(* if rst then *)
IF rst THEN
	piwl(rst := TRUE);
	piwl.RST := FALSE;
ELSE
	(* run PIWL controller first *)
	(* we need to check if TN = 0 and do alternative calls *)
	IF TN = 0.0 THEN
		piwl(in := IN * KP, KP := 1.0, KI := 0.0, LIM_L := LIM_L, LIM_H := LIM_H);
	ELSE
		piwl(in := IN * KP, KP := 1.0, KI := 1.0 / TN, LIM_L := LIM_L, LIM_H := LIM_H);
	END_IF;

	(* run differentiator and add_to_output *)
	diff(IN := IN, K := KP * TV);
	Y := piwl.Y + diff.out;
	(* add: output signal parts separately *)
	Y_p := piwl.Y_p;
	Y_i := piwl.Y_i;
	Y_d := diff.out;

	(* limit the output *)
	IF Y > LIM_H THEN
		Y := LIM_H;
		IF (Y_i > 0) THEN
			Y_i := LIM_H - Y_p - Y_d;
		END_IF
		LIM := TRUE;
	ELSIF Y < LIM_L THEN
		Y := LIM_L;
		IF (Y_i > 0) THEN
			Y_i := LIM_L - Y_p - Y_d;
		END_IF
		LIM := TRUE;
	ELSE
		LIM := FALSE;
	END_IF;
	
END_IF;



(* revision history
hm 13. jun. 2008 	rev 1.0
	original version

hm	25. jan 2008	rev 1.1
	multiply differential part with KP

hm	11. mar. 2009	rev 1.2
	real constants updated to new systax using dot

hm	13. nov. 2009	rev 1.3
	fixed code for negative KP

*)

END_FUNCTION_BLOCK

// A1_01A/Application/FUBs/Controller
// https://ftp.owen.ru/CoDeSys3/98_Books/oscat_basic333_ru.pdf		page 543, page 551
FUNCTION_BLOCK Controller
VAR_INPUT
	in: ctrl_input_typ;
	param: ctrl_param_typ;	
	cmd: ctrl_cmd_typ;
	cfg: UINT;
	t_move: UINT := 100;			// время на полную перестановку, сек (в текущей реализации как-то не у дел)
	t_error: UINT := 120;			// время на схождение положения крана и регулятора при регулировании
END_VAR
VAR_OUTPUT
	out: ctrl_output_typ;
	flags: ctrl_flags_typ;
END_VAR
VAR
	fub_pid: CTRL_PID;
	ton_diff: Standard.TON;
	ton_imit: Standard.TON;
END_VAR

(* Регулятор. 2 режима работы: стандартный, выход на ао
 * mode_manual - режим ручного ввода положения. управление аналоговое *)
		
IF cmd.manual_on THEN
	cmd.manual_on := FALSE;
	flags.mode_manual := TRUE;
END_IF
IF cmd.manual_off THEN
	cmd.manual_off := FALSE;
	flags.mode_manual := FALSE;
END_IF

IF cmd.imit_on THEN
	cmd.imit_on := FALSE;
	flags.mode_imit := TRUE;
	// при вкл имитации переведем пид в ручной режим на текущем уровне открытия и уставки
	in.man_value := in.im_pos_value := in.pos_value;
	in.set_value := in.act_value;
END_IF
IF cmd.imit_off THEN
	cmd.imit_off := FALSE;
	flags.mode_imit := FALSE;
END_IF

IF cmd.reset THEN
	cmd.reset := FALSE;
	flags.fail_open := FALSE;
	flags.fail_close := FALSE;
	flags.failed := FALSE;
END_IF
IF cmd.line_close THEN
	cmd.line_close := FALSE;
	IF flags.mode_imit THEN
		ton_imit.IN := TRUE;
		ton_imit.PT := REAL_TO_TIME( (UINT_TO_REAL(t_move) * in.im_pos_value/2/100)*1000 + 1);
	ELSE
		ton_imit.IN := FALSE;
		;// уставки приходится задавать снаружи (или встраивать alg_sp в пид)
	END_IF
END_IF
IF flags.mode_imit THEN
	in.pos_value := in.im_pos_value;
	// выход out_value не трогаем
	
	//IF b THEN
	ton_imit();
	//END_IF
	
	IF ton_imit.IN THEN
		in.im_pos_value := TIME_TO_REAL((ton_imit.PT - ton_imit.ET) / 1000 * 2);
	END_IF
	IF ton_imit.Q THEN
		ton_imit.IN := FALSE;
		in.im_pos_value := 0;
	END_IF
END_IF

fub_pid.ACT := in.act_value;
fub_pid.SET := in.set_value;
fub_pid.SUP := param.dead_zone;
fub_pid.OFS := param.offset;
fub_pid.M_I := in.man_value;
fub_pid.LL := param.min_out;
fub_pid.LH := param.max_out;
fub_pid.KP := param.k_p;
fub_pid.TN := param.t_i;
fub_pid.TV := param.t_d;
fub_pid.MAN := flags.mode_manual OR flags.mode_imit;
fub_pid();
out.err_value := fub_pid.DIFF;
out.out_value := fub_pid.Y;
out.p_part := fub_pid.Y_p;
out.i_part := fub_pid.Y_i;
out.d_part := fub_pid.Y_d;

flags.mode_dist := in.di_dist;
in.hyst_value := LIMIT(0.0, in.hyst_value, 5.0);
IF cfg.discrete_input THEN
	flags.open := in.di_open;
	flags.closed := in.di_closed;
ELSE
	flags.closed := in.pos_value <= in.hyst_value;
	flags.open := in.pos_value >= (100.0 - in.hyst_value);
END_IF

// Формирование команд дискретного управления регулирующим клапаном
flags.block_ao := NOT flags.mode_dist OR flags.mode_discrete OR flags.mode_manual OR flags.mode_imit;//cmd.line_close;
flags.ready := NOT in.di_fail AND flags.mode_dist AND NOT flags.block_ao; //исправим на NOT block_ao, потому что вообще нелогично

// Формирование сигнала «Неисправность регулирующего клапана»
ton_diff(IN := (param.discrepancy > 0.0 AND t_error > 0) AND_THEN ABS(in.pos_value - out.out_value) > (param.discrepancy + in.hyst_value) AND NOT flags.block_ao, PT := UDINT_TO_TIME(UINT_TO_UDINT(t_error) * 1000));
IF NOT flags.failed AND_THEN (in.di_fail OR ton_diff.Q OR flags.fail_open OR flags.fail_close) THEN
	flags.failed := TRUE;
	flags.mode_manual := TRUE;
END_IF

END_FUNCTION_BLOCK

// A1_01A/Application/Oscat/DEAD_ZONE
FUNCTION DEAD_ZONE : REAL
VAR_INPUT
	X : REAL;
	L : REAL;
END_VAR


(*
version 1.2	11. mar. 2009
programmer 	hugo
tested by		oscat

dead_zone2 is a linear transfer function which follows a linear function except for x is close to 0.
Y = X if abs(x) > L otherwise its 0.

*)

IF ABS(x) > L THEN
	dead_zone := X;
ELSE
	DEAD_ZONE := 0.0;
END_IF;

(* revision history
hm	12. feb. 2007	rev 1.0
	original version

hm	14. jun. 2008	rev 1.1
	improved performance

hm	11. mar. 2009	rev 1.2
	real constants updated to new systax using dot

*)

END_FUNCTION

// A1_01A/Application/Oscat/CTRL_PID
FUNCTION_BLOCK CTRL_PID
VAR_INPUT
	ACT : REAL;			// Значение регулируемой величины
	SET : REAL;			// Значение уставки
	SUP : REAL;			// Зона нечувствительности
	OFS : REAL;			// Смещение
	M_I : REAL;			// Значение ручного ввода
	MAN : BOOL;			// Сигнал ручного ввода
	RST : BOOL;			// Сигнал обнуления И-составляющей
	KP : REAL := 1.0;
	TN : REAL := 1.0;
	TV : REAL := 1.0;
	LL : REAL := -1000.0;	// Нижний предел управляющего сигнала
	LH : REAL := 1000.0;	// Верхний предел управляющего сигнала
END_VAR
VAR_OUTPUT
	Y : REAL;			// Величина управляющего воздействия
	Y_p : REAL;
	Y_i : REAL;
	Y_d : REAL;
	DIFF : REAL;		// Сигнал рассогласования
	LIM : BOOL;			// Флаг «достигнут предел для Y»
END_VAR
VAR
	pid : FT_PIDWL;
	co : CTRL_OUT;
END_VAR



(*
version 2.0	30. jun. 2008
programmer 	hugo
tested by	oscat

FT_PI is a PI controller with manual functionality.
The PID controller works according to the fomula Y = e *(KP+ KI * INTEG(e) ) + offset, while e = set_point - actual.
a rst will reset all internal data, while a switch to manual will cause the controller to follow the function Y = manual_in + offset.
limit_h and Limit_l set the possible output range of Y.
the output flags lim will signal that the output limits are active.

*)

DIFF := CTRL_IN(SET, ACT, SUP);
pid(in := DIFF, kp := KP, tn := TN, tv := TV, lim_l := LL, lim_h := LH, rst := RST);
co(ci := pid.Y, OFFSET := OFS, man_in := M_I, lim_l := LL, lim_h := LH, MANUAL := MAN);
Y := co.Y;
LIM := co.LIM;

Y_p := pid.Y_p;
Y_i := pid.Y_i;
Y_d := pid.Y_d;

(* revision history

hm 1.12.2006	 	rev 1.1
	changed algorithm to trapezregel for higher accuracy.

hm 3.1.2007		rev 1.2
	added integ_band to select when the integrator is active.

hm	3.3.2007		rev 1.3
	added default values to inputs KP, TN, TV, LIMIT_L und LIMIT_H.

hm 31.oct 2007	rev 1.4
	total rewrite of the module to avoid failures when one of the limits is 0

hm	3.11.2007	rev 1.5
	added noise input to filter noise
	added output diff
	set limit output false when output is within limits
	overfolw was not set correctly

hm	5. jan 2008	rev 1.6
	improved code for better performance
*)

END_FUNCTION_BLOCK

// A1_01A/Application/Oscat/CTRL_IN
FUNCTION CTRL_IN : REAL
VAR_INPUT
	SET_POINT, ACTUAL, NOISE : REAL;
END_VAR


(*
version 1.0	2. jun 2008
programmer 	hugo
tested by		tobias


*)

(* calculate the process error DIFF *)
CTRL_IN := DEAD_ZONE(SET_POINT - ACTUAL, NOISE);


(* revision history
hm 	2. jun. 2008 	rev 1.0
	original version

*)

END_FUNCTION

// A1_01A/Application/Oscat/FT_PIWL
FUNCTION_BLOCK FT_PIWL
VAR_INPUT
	IN : REAL;
	KP : REAL := 1.0;
	KI : REAL := 1.0;
	LIM_L : REAL := -1.0E38;
	LIM_H : REAL := 1.0E38;
	RST : BOOL;
END_VAR
VAR_OUTPUT
	Y : REAL;
	Y_p : REAL;
	Y_i : REAL;
	LIM : BOOL;
END_VAR
VAR
	init: BOOL;
	tx: DWORD;
	tc : REAL;
	t_last: DWORD;
	in_last : REAL;
	i: REAL;
	p: REAL;
END_VAR

(*
version 1.3	11. mar. 2009
programmer 	hugo
tested by		oscat

FT_PIWL is a PI controller.
The PID controller works according to the fomula Y = IN *(KP+ KI * INTEG(e) ).
a rst will reset the integrator to 0
lim_h and Lim_l set the possible output range of the controller.
the output flag lim will signal that the output limits are active.
the integrator ist equipped with anti wind-up circuitry which limits trhe total output ranke to lim_l and lim_h

default values for KP = 1, KI = 1, ILIM_L = -1E37, iLIM_H = +1E38.
*)

(* initialize at power_up *)
IF NOT init OR RST THEN
	init := TRUE;
	in_last := in;
	t_last := T_PLC_US();
	i := 0.0;
	tc := 0.0;
ELSE
	(* read last cycle time in Microseconds *)
	tx := T_PLC_US();
	tc := DWORD_TO_REAL(tx - t_last);
	t_last := tx;

	(* calculate proportional part *)
	p := KP * IN;

	(* run integrator *)
	i := (IN + in_last) * 5.0E-7 * KI * tc + i;
	in_last := IN;

	(* calculate output Y *)
	Y := p + i;

	(* check output for limits *)
	IF Y >= LIM_H THEN
		Y := LIM_H;
		IF ki <> 0.0 THEN
			i := LIM_H - p;
		ELSE
			i := 0.0;
		END_IF;
		LIM := TRUE;
	ELSIF Y <= LIM_L THEN
		Y := LIM_L;
		IF ki <> 0.0 THEN
			i := LIM_L - p;
		ELSE
			i := 0.0;
		END_IF;
		LIM := TRUE;
	ELSE
		LIM := FALSE;
	END_IF;
	
	(* add: output signal parts separately *)
	Y_p := p;
	Y_i := i;
END_IF;




(* revision history
hm 13. jun. 2008 	rev 1.0
	original version

hm	27. oct. 2008	rev 1.1
	integrator will not be adjusted when ki = 0

hm	25. jan 2009	rev 1.2
	module will also work with negative K

hm	11. mar. 2009	rev 1.3
	real constants updated to new systax using dot

*)

END_FUNCTION_BLOCK

// A1_01A/Application/Oscat/FT_DERIV
FUNCTION_BLOCK FT_DERIV
VAR_INPUT
	in : REAL;
	K : REAL := 1.0;
	run : BOOL := TRUE;
END_VAR
VAR_OUTPUT
	out : REAL;
END_VAR
VAR
	old: REAL;
	tx: DWORD;
	last: DWORD;
	init: BOOL;
	tc: REAL;
END_VAR


(*
version 1.5	11. mar. 2009
programmer 	hugo
tested by		oscat

FT_deriv calculates the derivate over the signal "in" with Faktor "K".
a run input enables or stops the calculation, if left unconnected its true and therfore the calculation is executed.
if K is not specified the default is 1.

*)

(* read system time *)
tx := T_PLC_US();
tc := DWORD_TO_REAL(tx - last);
last := tx;

(* init on first startup *)
IF NOT init THEN
	init := TRUE;
	old := in;
ELSIF run AND tc > 0.0 THEN
	out := (in - old) / tc * 1000000.0 * K;
	old := in;
ELSE
	out := 0.0;
END_IF;



(*
hm 3.1.2007			rev 1.1
	added init code for startup
	set the default for K to 1

hm	15. sep 2007	rev 1.2
	replaced Time() with T_PLC_US for compatibility and performance reasons
	increased accuracy and work in microseconds internally

hm 29 oct 2007	rev 1.3
	prohibit calculation when tx - last = 0 to avoid division by 0 and increase accuracy on fast systems

hm	6. nov. 2008	rev 1.4
	improved performance

hm	11. mar. 2009	rev 1.5
	inproved code
*)

END_FUNCTION_BLOCK

// A1_01A/Application/FUBs/LineMeteringRLT
FUNCTION_BLOCK LineMeteringRLT	// Алгоритм нитки расхода
VAR_INPUT
	num_v_in, num_v_out: UINT;	// номера кранов из массива на входе/выходе этой нитки
	param: line_param_f_typ;
	cmd: line_cmd_typ;			// прямые команды управления 
	a_in: line_act_in;			// внешнее алгоритмическое управление
	a_out: line_act_out;		// результат исполнения
	flow_online: BOOL;			// расходомер на связи, расход актуален
	busy: BOOL;					// нитка занята в алгоритме
	a_to: USINT;				// номер нитки, в которую была выдана команда
END_VAR
VAR_OUTPUT
	flags: line_flags_f_typ;
END_VAR
VAR
END_VAR

IF cmd.block_on THEN
	cmd.block_on := FALSE;
	flags.mode_block := TRUE;
END_IF
IF cmd.block_off THEN
	cmd.block_off := FALSE;
	flags.mode_block := FALSE;
END_IF
IF cmd.manual_on THEN
	cmd.manual_on := FALSE;
	flags.mode_manual := TRUE;
END_IF
IF cmd.manual_off THEN
	cmd.manual_off := FALSE;
	flags.mode_manual := FALSE;
END_IF
IF cmd.reset THEN
	cmd.reset := FALSE;
	flags.failed := FALSE;
	flags.fail_block := FALSE;
END_IF
IF (flags.mode_block AND (a_in.a_cmd > 0 OR cmd.open OR cmd.close)) THEN
	a_in.a_cmd := en_line_action.LA_NONE;
	a_in.a_from := -1;
	cmd.open := FALSE;
	cmd.close := FALSE;
	flags.fail_block := TRUE;
END_IF

IF num_v_in < COUNT_VALVE AND num_v_out < COUNT_VALVE THEN
	flags.err_num := FALSE;
	flags.open := sys_valve[num_v_in].v_state = RLTAB.en_valve_state.VALVESTT_OPEN AND sys_valve[num_v_out].v_state = RLTAB.en_valve_state.VALVESTT_OPEN;
	flags.closed := sys_valve[num_v_in].v_state = RLTAB.en_valve_state.VALVESTT_CLOSED AND sys_valve[num_v_out].v_state = RLTAB.en_valve_state.VALVESTT_CLOSED;
	flags.ready := (sys_valve[num_v_in].flags.ready AND sys_valve[num_v_out].flags.ready) AND NOT flags.mode_block;
	// T6.1,141 Формирование сигнала о неисправности линии редуцирования
	// VALVE: flags.ready := (v_mode > MODE_BUTTON) AND NOT flags.mode_block AND NOT (flags.cv_fail OR flags.fail_open OR flags.fail_close);
	IF flags.open AND NOT flags.ready AND NOT flags.mode_reserve THEN
		flags.failed := TRUE;
	END_IF
	
	IF flags.mode_manual THEN
		param.flow_actual := param.flow_manual;
	END_IF
	IF flags.open AND param.flow_lo <> param.flow_hi THEN
		IF param.flow_actual < (param.flow_lo - param.flow_hyst) THEN
			flags.flow_lo := TRUE;
			flags.flow_ok := FALSE;
		ELSIF param.flow_actual > (param.flow_lo + param.flow_hyst) THEN
			flags.flow_lo := FALSE;
			flags.flow_ok := TRUE;
		END_IF
		IF param.flow_actual > (param.flow_hi + param.flow_hyst) THEN
			flags.flow_hi := TRUE;
			flags.flow_ok := FALSE;
		ELSIF param.flow_actual < (param.flow_hi - param.flow_hyst) THEN
			flags.flow_hi := FALSE;
			flags.flow_ok := TRUE;
		END_IF
	ELSE
		flags.flow_lo := FALSE;
		flags.flow_ok := FALSE;
		flags.flow_hi := FALSE;
	END_IF
		
	// лучше использовать эти команды a_in для внешнего алгоритмического управления, т.к. в них встроена защита от busy
	IF a_in.a_cmd > 0 THEN
		a_out.done := FALSE;
		IF a_out.result <> en_line_action.LA_BUSY (*AND NOT flags.mode_block*) THEN
			a_out.a_orig := a_in.a_cmd;
			//a_in.a_cmd := en_line_action.LA_NONE;
			a_out.a_from := a_in.a_from;
			//a_in.a_from := -1;
			CASE a_out.a_orig OF
				en_line_action.LA_OPEN:
					cmd.open := TRUE;
				en_line_action.LA_CLOSE:
					cmd.close := TRUE;
			END_CASE
			a_out.result := en_line_action.LA_BUSY;
		END_IF
		a_in.a_cmd := en_line_action.LA_NONE;
		a_in.a_from := -1;
	END_IF
	IF a_out.result = en_line_action.LA_BUSY THEN
		CASE a_out.a_orig OF
			en_line_action.LA_OPEN:
				IF flags.ready THEN
					IF flags.open THEN
						a_out.result := en_line_action.LA_OPEN;
						a_out.done := TRUE;
					END_IF
				ELSE
					a_out.result := en_line_action.LA_ERROR;
					a_out.done := TRUE;
				END_IF
				
			en_line_action.LA_CLOSE:
				IF flags.ready THEN
					IF flags.closed THEN
						a_out.result := en_line_action.LA_CLOSE;
						a_out.done := TRUE;
					END_IF
				ELSE
					a_out.result := en_line_action.LA_ERROR;
					a_out.done := TRUE;
				END_IF
				
		END_CASE
	END_IF
	
	IF cmd.open THEN
		cmd.open := FALSE;
		sys_valve[num_v_in].cmd.open := TRUE;
		sys_valve[num_v_out].cmd.open := TRUE;
	END_IF
	IF cmd.close THEN
		cmd.close := FALSE;
		sys_valve[num_v_in].cmd.close := TRUE;
		sys_valve[num_v_out].cmd.close := TRUE;
	END_IF
ELSE
	flags.err_num := TRUE;
	flags.open := FALSE;
	flags.closed := FALSE;
	flags.ready := FALSE;
	a_in.a_cmd := en_line_action.LA_NONE;
	a_in.a_from := -1;
	cmd.open := FALSE;
	cmd.close := FALSE;
END_IF

METHOD Init
VAR_INPUT
	value: BOOL;
END_VAR
THIS^.flags.mode_reserve := value;
END_METHOD

METHOD _set_mr
VAR_INPUT
	value: BOOL;
END_VAR
THIS^.flags.mode_reserve := value;
END_METHOD

END_FUNCTION_BLOCK

// A1_01A/Application/FUBs/LineReducingRLT
FUNCTION_BLOCK LineReducingRLT	// Алгоритм нитки редуцирования
VAR_INPUT
	num_ctrl: UINT;				// номер ПИДа на этой нитки
	num_v_in, num_v_out: UINT;	// номера кранов из массива на входе/выходе этой нитки
	cmd: line_cmd_typ;			// прямые команды управления 
	a_in: line_act_in;			// внешнее алгоритмическое управление
	a_out: line_act_out;		// результат исполнения
	busy: BOOL;					// нитка занята в алгоритме
	a_to: USINT;				// номер нитки, в которую была выдана команда
END_VAR
VAR_OUTPUT
	flags: line_flags_r_typ;
END_VAR
VAR
END_VAR

IF cmd.block_on THEN
	cmd.block_on := FALSE;
	flags.mode_block := TRUE;
END_IF
IF cmd.block_off THEN
	cmd.block_off := FALSE;
	flags.mode_block := FALSE;
END_IF
IF cmd.reset THEN
	cmd.reset := FALSE;
	flags.failed := FALSE;
	flags.fail_block := FALSE;
END_IF
IF (flags.mode_block AND (a_in.a_cmd > 0 OR cmd.open OR cmd.close)) THEN
	a_in.a_cmd := en_line_action.LA_NONE;
	a_in.a_from := -1;
	cmd.open := FALSE;
	cmd.close := FALSE;
	flags.fail_block := TRUE;
END_IF

IF num_v_in < COUNT_VALVE AND num_ctrl < CFGCONST.COUNT_LINES AND num_v_out < COUNT_VALVE THEN
	flags.err_num := FALSE;
	flags.open := sys_valve[num_v_in].v_state = RLTAB.en_valve_state.VALVESTT_OPEN AND sys_valve[num_v_out].v_state = RLTAB.en_valve_state.VALVESTT_OPEN;
	flags.closed := sys_valve[num_v_in].v_state = RLTAB.en_valve_state.VALVESTT_CLOSED AND pid[num_ctrl].flags.closed AND sys_valve[num_v_out].v_state = RLTAB.en_valve_state.VALVESTT_CLOSED;
	flags.ready := (sys_valve[num_v_in].flags.ready AND pid[num_ctrl].flags.ready AND sys_valve[num_v_out].flags.ready) AND NOT flags.mode_block;
	// T6.1,141 Формирование сигнала о неисправности линии редуцирования
	// VALVE: flags.ready := (v_mode > MODE_BUTTON) AND NOT flags.mode_block AND NOT (flags.cv_fail OR flags.fail_open OR flags.fail_close);
	IF flags.open AND NOT flags.ready AND NOT flags.mode_reserve THEN
		flags.failed := TRUE;
	END_IF
	
	// лучше использовать эти команды a_in для внешнего алгоритмического управления, т.к. в них встроена защита от busy
	IF a_in.a_cmd > 0 THEN
		a_out.done := FALSE;
		IF a_out.result <> en_line_action.LA_BUSY (*AND NOT flags.mode_block*) THEN
			a_out.a_orig := a_in.a_cmd;
			//a_in.a_cmd := en_line_action.LA_NONE;
			a_out.a_from := a_in.a_from;
			//a_in.a_from := -1;
			CASE a_out.a_orig OF
				en_line_action.LA_OPEN:
					cmd.open := TRUE;
				en_line_action.LA_CLOSE:
					cmd.close := TRUE;
			END_CASE
			a_out.result := en_line_action.LA_BUSY;
		END_IF
		a_in.a_cmd := en_line_action.LA_NONE;
		a_in.a_from := -1;
	END_IF
	IF a_out.result = en_line_action.LA_BUSY THEN
		CASE a_out.a_orig OF
			en_line_action.LA_OPEN:
				IF flags.ready THEN
					IF flags.open THEN
						a_out.result := en_line_action.LA_OPEN;
						a_out.done := TRUE;
					END_IF
				ELSE
					a_out.result := en_line_action.LA_ERROR;
					a_out.done := TRUE;
				END_IF
				
			en_line_action.LA_CLOSE:
				IF flags.ready THEN
					IF flags.closed THEN
						a_out.result := en_line_action.LA_CLOSE;
						a_out.done := TRUE;
					END_IF
				ELSE
					a_out.result := en_line_action.LA_ERROR;
					a_out.done := TRUE;
				END_IF
				
		END_CASE
	END_IF
	
	IF cmd.open THEN
		cmd.open := FALSE;
		sys_valve[num_v_in].cmd.open := TRUE;
		pid[num_ctrl].cmd.manual_off := TRUE;
		sys_valve[num_v_out].cmd.open := TRUE;
	END_IF
	IF cmd.close THEN
		cmd.close := FALSE;
		sys_valve[num_v_in].cmd.close := TRUE;
		pid[num_ctrl].cmd.line_close := TRUE;
		pid[num_ctrl].cmd.manual_on := TRUE;
		sys_valve[num_v_out].cmd.close := TRUE;
	END_IF
ELSE
	flags.err_num := TRUE;
	flags.open := FALSE;
	flags.closed := FALSE;
	flags.ready := FALSE;
	a_in.a_cmd := en_line_action.LA_NONE;
	a_in.a_from := -1;
	cmd.open := FALSE;
	cmd.close := FALSE;
END_IF

METHOD Init
VAR_INPUT
	value: BOOL;
END_VAR
THIS^.flags.mode_reserve := value;
END_METHOD

METHOD _set_mr
VAR_INPUT
	value: BOOL;
END_VAR
THIS^.flags.mode_reserve := value;
END_METHOD

END_FUNCTION_BLOCK

// A1_01A/Application/FUBs/LineGroupRLT
FUNCTION_BLOCK LineGroupRLT			// Алгоритм управления группой ниток по аналогам БАКСа
VAR_INPUT							// поддерживает LineReducingRLT и LineMeteringRLT без доработок через объявление в GVL
	lines: ARRAY [0..COUNT_LINES-1] OF UINT;	// номера ниток в группе 0..max-1
	count: UINT := CFGCONST.COUNT_LINES;		// кол-во ниток, макс все в одной группе 
	cmd: line_cmd_grp_typ;
	
	new_res_line: UINT;				// новая резервная нитка
	lines_needed: USINT;			// сколько ниток требуется
	t_change: UINT := 30;			// время на перестановку линии, сек
	enable: BOOL;
	automatic: BOOL;				// включен автоматический режим
	stop_now: BOOL;					// немедленно все закрыть
END_VAR
VAR_OUTPUT
	lines_at_work: USINT;			// столько ниток в работе
	old_res_line: UINT;				// текущая резервная нитка
	// алгоритм: смена резервной нитки
	line_reserve_want: BOOL;		// алгоритм хочет запустится, но нитки еще заняты другим
	line_reserve_run: BOOL;			// алгоритм работает
	line_reserve_fail: BOOL;		// авария алгоритма
	// алгоритм: переключение ниток по аварии
	line_fault_block: BOOL;			// алгоритм заблокирован
	line_fault_want: BOOL;
	line_fault_run: BOOL;
	line_fault_fail: BOOL;
	// алгоритм: управление нитками по расходу
	line_flow_block: BOOL;
	line_flow_want: BOOL;
	line_flow_run: BOOL;
	line_flow_no_open: BOOL;		// нет нитки для открытия
	line_flow_no_close: BOOL;		// нет нитки для закрытия
END_VAR
VAR
	ton_res: Standard.TON;
	ton_fault: Standard.TON;
	ton_flow: Standard.TON;
	i, j, n: USINT;
	b, v: BOOL;
END_VAR

IF NOT enable THEN
	RETURN;
END_IF
IF count > CFGCONST.COUNT_LINES THEN
	count := CFGCONST.COUNT_LINES;
END_IF
//	в принципе эти алгоритмы подходят для любых ниток с похожим интерейсом. можно переделать через него...
//	управление: count, new_res_line, lines_needed, у ниток: cmd, flags

IF cmd.block_fault_on THEN
	cmd.block_fault_on := FALSE;
	line_fault_block := TRUE;
END_IF
IF cmd.block_fault_off THEN
	cmd.block_fault_off := FALSE;
	line_fault_block := FALSE;
END_IF
IF cmd.block_flow_on THEN
	cmd.block_flow_on := FALSE;
	line_flow_block := TRUE;
END_IF
IF cmd.block_flow_off THEN
	cmd.block_flow_off := FALSE;
	line_flow_block := FALSE;
END_IF
IF stop_now THEN
	line_fault_block := TRUE;
	line_flow_block := TRUE;
END_IF

IF cmd.close THEN
	IF NOT line_reserve_run AND NOT line_reserve_run AND NOT line_flow_run THEN
		cmd.close := FALSE;
		FOR i := 0 TO CFGCONST.COUNT_LINES-1 DO
			line[i].a_in.a_cmd := en_line_action.LA_CLOSE;
			line[i].a_in.a_from := 0;
		END_FOR
	END_IF
END_IF
IF cmd.reset THEN
	cmd.reset := FALSE;
	line_reserve_fail := FALSE;
	line_fault_fail := FALSE;
	line_flow_no_open := FALSE;
	line_flow_no_close := FALSE;
	FOR i := 0 TO CFGCONST.COUNT_LINES-1 DO
		line[i].cmd.reset := TRUE;
	END_FOR
END_IF

// ПОКА ЧТО оставим захардкоженные линии 6 штук. подумать как присвоить их потом
lines_at_work := 0;
FOR i := 0 TO CFGCONST.COUNT_LINES-1 DO
	line[i]();
	lines_at_work := lines_at_work + BOOL_TO_USINT(line[i].flags.open);
END_FOR

// общее: начинаем общий алгоритм если ничего другого не исполняется и если нет блока
// но если уже работает, должен дойти до конца

// Алгоритм: смена резервной нитки
IF new_res_line <> old_res_line AND NOT line_reserve_fail AND NOT line_reserve_run THEN	// "AND NOT line_reserve_run" здесь не особо обязателен, т.к. есть в IF ниже. но "заход" тогда все равно пустой получается
	IF automatic AND NOT stop_now AND NOT line_fault_run AND NOT line_flow_run THEN
		//IF NOT line_reserve_run THEN
			line_reserve_run := TRUE;
			line_reserve_want := FALSE;
		//END_IF
	ELSE
		line_reserve_want := TRUE;
	END_IF
ELSE
	line_reserve_want := FALSE;
END_IF
ton_res(IN := line_reserve_run, PT := UDINT_TO_TIME(UINT_TO_UDINT(t_change) * 1000));
IF line_reserve_run THEN
	IF NOT line[old_res_line].flags.ready OR NOT line[new_res_line].flags.ready OR ton_res.Q THEN		// flags.failed ? в ready включены аварии кранов, но оно сбрасывается само
		// в данном случае ошибки кранов включены в флаг ready, поэтому так норм
		line_reserve_run := FALSE;
		//old_res_line := new_res_line;
		line_reserve_fail := TRUE;
	ELSIF line[old_res_line].flags.closed AND line[new_res_line].flags.closed THEN
		line_reserve_run := FALSE;
		line[old_res_line]._set_mr(FALSE);
		line[new_res_line]._set_mr(TRUE);
		old_res_line := new_res_line;
	ELSE
		// откроем новую линию, затем закроем старую. после завершения поменяем статусы
		IF NOT line[old_res_line].flags.open THEN
			line[old_res_line].a_in.a_cmd := en_line_action.LA_OPEN;
			line[old_res_line].a_in.a_from := 0;
		END_IF
		IF line[old_res_line].flags.open AND line[old_res_line].a_out.done AND NOT line[new_res_line].flags.closed THEN
			line[old_res_line].a_out.done := FALSE;
			line[new_res_line].a_in.a_cmd := en_line_action.LA_CLOSE;
			line[new_res_line].a_in.a_from := 0;
		END_IF
		IF line[old_res_line].flags.open AND line[new_res_line].flags.closed AND line[new_res_line].a_out.done THEN
			line[new_res_line].a_out.done := FALSE;
			line[old_res_line]._set_mr(FALSE);
			line[new_res_line]._set_mr(TRUE);
			old_res_line := new_res_line;
			line_reserve_run := FALSE;
		END_IF
		
	END_IF
END_IF

// алгоритм: смена нитки по аварии
b := FALSE;
FOR i := 0 TO CFGCONST.COUNT_LINES-1 DO
	IF line[i].flags.failed AND NOT line[i].flags.mode_block AND NOT line[i].busy AND NOT line_fault_block AND NOT line_fault_fail THEN	// добавим mode_block чтобы срабатывало 1 раз. /failed подразумевает open
		IF automatic AND NOT stop_now (*AND NOT line_fault_block*) AND NOT line_reserve_run AND NOT line_flow_run THEN					// правильнее R_TRIG на аварию, но ломаются приоритеты вычисления т.к. оно снаружи
			line_fault_run := TRUE;
			line_fault_want := FALSE;
		ELSE
			//line_fault_want := FALSE;
			b := b OR TRUE;
		END_IF
	//ELSE
	//	line_fault_want := FALSE;
	END_IF
END_FOR
line_fault_want := b;
ton_fault(IN := line_fault_run, PT := UDINT_TO_TIME(UINT_TO_UDINT(t_change) * 1000));
IF line_fault_run THEN
	FOR i := 0 TO CFGCONST.COUNT_LINES-1 DO
		// линия в аварии и еще не обрабатывается
		IF line[i].flags.failed AND NOT line[i].flags.mode_block AND NOT line[i].busy THEN	// flags.closed использовать нельзя, т.к. нет гарантии что оно закроется
			n := i; b := FALSE; v := FALSE;
			// поиск доступной не открытой не занятой нитки
			FOR j := 1 TO CFGCONST.COUNT_LINES-1 DO
				n := _next(n);
				IF line[n].flags.ready AND NOT line[n].flags.mode_reserve AND NOT line[n].flags.open THEN
					v := TRUE;	// если есть подходящая нитка, но она пока занята
					IF NOT line[n].busy THEN
						b := TRUE; EXIT;
					END_IF
				END_IF
			END_FOR
			// подходящая нитка найдена - открыть
			IF b THEN
				line[i].busy := TRUE;
				line[i].a_to := n;	// сохраняем что аварийная нитка хочет открыть N
				line[n].busy := TRUE;
				line[n].a_in.a_cmd := en_line_action.LA_OPEN;
				line[n].a_in.a_from := USINT_TO_SINT(i);
			ELSIF NOT v THEN
				// нитка не найдена
				line_fault_fail := TRUE;
				// run не снимаем, чтобы если есть текущие нитки, они могли завершить свою операцию. после этого он снимется сам.
			END_IF
		END_IF
	END_FOR
	
	b := FALSE;
	FOR i := 0 TO CFGCONST.COUNT_LINES-1 DO
		b := b OR line[i].busy;
		IF line[i].flags.failed AND NOT line[i].flags.mode_block AND line[i].busy THEN
			n := line[i].a_to;
			// проверяем что нитки в норме
			IF NOT line[n].flags.ready OR NOT line[i].flags.ready OR ton_fault.Q THEN
				line[i].busy := FALSE;
				line[n].busy := FALSE;
				line_fault_fail := TRUE;
			ELSE
				// открываем новую нитку и закрываем старую
				IF line[n].flags.open AND line[n].a_out.done AND NOT line[i].flags.closed THEN
					line[n].a_out.done := FALSE;
					line[i].a_in.a_cmd := en_line_action.LA_CLOSE;
					line[i].a_in.a_from := 0;
				END_IF
				IF line[n].flags.open AND line[i].flags.closed AND line[i].a_out.done THEN
					line[i].a_out.done := FALSE;
					line[i].busy := FALSE;
					line[n].busy := FALSE;
					line[i].cmd.block_on := TRUE;
				END_IF
				
			END_IF // !r & !r
		END_IF //f & b
	END_FOR
	
	line_fault_run := b;
END_IF

// алгоритм: управление нитками по расходу
IF ton_flow.Q THEN
	line[n].busy := FALSE;
	line_flow_run := FALSE;
	ton_flow.IN := FALSE;
	ton_flow();
END_IF
IF lines_needed <> lines_at_work AND NOT line_flow_run THEN											// разница "NOT line_flow_run" и "NOT line[i].busy" в том, что в 1. мы проверяем алгоритм запущен вообще
	IF automatic AND NOT stop_now AND NOT line_flow_block AND NOT line_reserve_run AND NOT line_fault_run THEN	// а в 2. алгоритм может быть запущен по нескольким ниткам одновременно и проверяем каждую
		IF line_flow_no_open OR line_flow_no_close THEN		// если были ошибки
			line_flow_want := TRUE;
		END_IF
		IF lines_needed > lines_at_work AND NOT line_flow_no_open THEN
			line_flow_run := TRUE;
			line_flow_want := FALSE;
		END_IF
		IF lines_needed < lines_at_work AND NOT line_flow_no_close THEN
			line_flow_run := TRUE;
			line_flow_want := FALSE;
		END_IF
	ELSE
		line_flow_want := TRUE;
	END_IF
ELSE
	line_flow_want := FALSE;
END_IF
IF line_flow_run AND NOT ton_flow.IN THEN
	// проверка на ready наверное не нужна, т.к. включена в поиске ниток, а если их не было найдено и так возникнет ошибка
	IF lines_needed > lines_at_work (*AND NOT line_flow_no_open*) THEN
		b := FALSE;
		FOR i := 0 TO CFGCONST.COUNT_LINES-1 DO		// можно переделать на цикл через _next, тогда нитки будут переключаться по очереди вместо всегда первой.
			IF line[i].flags.ready AND NOT line[i].flags.mode_reserve AND NOT line[i].flags.open THEN
				n := i; b := TRUE; EXIT;
			END_IF
		END_FOR
		IF b THEN
			//line[n].busy := TRUE;		а где снимать busy?
			line[n].a_in.a_cmd := en_line_action.LA_OPEN;
			line[n].a_in.a_from := USINT_TO_SINT(n);
		ELSE
			line_flow_no_open := TRUE;
		END_IF
	END_IF
	IF lines_needed < lines_at_work (*AND NOT line_flow_no_close*) THEN
		b := FALSE;
		FOR i := 0 TO CFGCONST.COUNT_LINES-1 DO
			IF line[i].flags.ready AND NOT line[i].flags.mode_reserve AND NOT line[i].flags.closed THEN
				n := i; b := TRUE; EXIT;
			END_IF
		END_FOR
		IF b THEN
			//line[n].busy := TRUE;
			line[n].a_in.a_cmd := en_line_action.LA_CLOSE;
			line[n].a_in.a_from := USINT_TO_SINT(n);
		ELSE
			line_flow_no_close := TRUE;
		END_IF
	END_IF
	ton_flow.IN := TRUE;	// запуск таймера, алгоритм продолжится после установления режима
END_IF
ton_flow(PT := UDINT_TO_TIME(UINT_TO_UDINT(t_change) * 1000));

// алгоритм: аварийный останов - отдельно оказалось не надо

METHOD Init
VAR_INPUT
	num: UINT;
END_VAR
VAR
	i: UINT;
END_VAR
THIS^.new_res_line := THIS^.old_res_line := num;
FOR i := 0 TO CFGCONST.COUNT_LINES-1 DO
	line[i].Init(FALSE);
END_FOR
line[num].Init(TRUE);
END_METHOD

METHOD PRIVATE _next : USINT
VAR_INPUT
	num: USINT;
END_VAR
IF num < CFGCONST.COUNT_LINES(*count*)-1 THEN
	_next := num + 1;
ELSE
	_next := 0;
END_IF
END_METHOD

END_FUNCTION_BLOCK

// A1_01A/Application/Devices/V_Ope_TM
FUNCTION_BLOCK V_Ope_TM EXTENDS RLTM.DeviceTemplate
VAR_INPUT
END_VAR
VAR_OUTPUT
	tf: ARRAY[0..21] OF RLTNU.IEC_M_ME_NC;
END_VAR
VAR
	data_real: ARRAY[0..21] OF REAL;
	res: ARRAY[0..9] OF RLTM.RLTM_MODBUS_TRANSACTION_RESULT;
	i, j: UINT;
	c: ARRAY[0..15] OF UINT := [ 16#1, 16#2, 16#4, 16#8, 16#10, 16#20, 16#40, 16#80, 16#100, 16#200, 16#400, 16#800, 16#1000, 16#2000, 16#4000, 16#8000 ];
END_VAR

(*
Мгновенная активная мощность по фазе 1
Мгновенная активная мощность по фазе 2
Мгновенная активная мощность по фазе 3
Напряжение по фазе 1
Напряжение по фазе 2
Напряжение по фазе 3
Ток по фазе 1
Ток по фазе 2
Ток по фазе 3
Суммарная активная мощность от сброса
Суммарная активная мощность до сброса
Суммарная реактивная мощность от сброса
Суммарная реактивная мощность до сброса
Активная мощность от сброса за текущие сутки
Активная мощность до сброса за текущие сутки
Реактивная мощность от сброса за текущие сутки
Реактивная мощность до сброса за текущие сутки
Активная мощность от сброса за предыдущие сутки
Активная мощность до сброса за предыдущие сутки
Реактивная мощность от сброса за предыдущие сутки
Реактивная мощность до сброса за предыдущие сутки
*)
FOR i := 0 TO 0 DO
	CASE res[i] OF
		RLTM.RLTM_TRANSACTION_RESULT_PROCESSING:
			;//nothing to do
		RLTM.RLTM_TRANSACTION_RESULT_SUCCESS:
			CASE i OF
				0:
					FOR j := 0 TO 21 DO
						tf[j].value := data_real[j];
						tf[j].qds.b.IV := 0;
					END_FOR
				
			END_CASE
	ELSE
		CASE i OF
				0:
					FOR j := 0 TO 21 DO
						tf[j].qds.b.IV := 1;
					END_FOR
		END_CASE
	END_CASE
END_FOR

METHOD Init: BOOL;
VAR_INPUT
END_VAR
VAR

END_VAR
SUPER^.Init();
transaction.typ := RLTM.RLTM_TRANSACTION_TYP_DATA;
transaction.mfc := 3;
transaction.offset := 0;
transaction.len := 42;
transaction.swap_byte := 1;
transaction.pData := ADR(data_real[0]);
transaction.pRes := ADR(res[0]);
transaction.timer.PT := T#1S;
SUPER^.AppendTransaction();

Init := 1;
END_METHOD

END_FUNCTION_BLOCK

// A1_01A/Application/Devices/EK
FUNCTION_BLOCK EK EXTENDS RLTM.DeviceTemplate
VAR_INPUT
END_VAR
VAR_OUTPUT
	tf: ARRAY[0..21] OF RLTNU.IEC_M_ME_NC;
END_VAR
VAR
	data_real: ARRAY[0..21] OF REAL;
	res: ARRAY[0..9] OF RLTM.RLTM_MODBUS_TRANSACTION_RESULT;
	i, j: UINT;
	c: ARRAY[0..15] OF UINT := [ 16#1, 16#2, 16#4, 16#8, 16#10, 16#20, 16#40, 16#80, 16#100, 16#200, 16#400, 16#800, 16#1000, 16#2000, 16#4000, 16#8000 ];
END_VAR

(*
Давление
Температура
Абсолютное давление
Коэффициент коррекции 
Коэффициент сжимаемости газа
Содержание азота
Содержание водорода
Содержание двуокиси углерода
Плость газа при нормальных условиях
Рабочий расход газа
Стандартный расход газа
Мощность
Теплотворная способность
Коэффициент плотности
Давление
Температура
Рабочий объём
Стандартный объём
Энергия
Рабочий расход прошлые сутки
Стандартный расход прошлые сутки
Рабочий расход прошлый месяц
Стандартный расход прошлый месяц
*)
FOR i := 0 TO 0 DO
	CASE res[i] OF
		RLTM.RLTM_TRANSACTION_RESULT_PROCESSING:
			;//nothing to do
		RLTM.RLTM_TRANSACTION_RESULT_SUCCESS:
			CASE i OF
				0:
					FOR j := 0 TO 23 DO
						tf[j].value := data_real[j];
						tf[j].qds.b.IV := 0;
					END_FOR
				
			END_CASE
	ELSE
		CASE i OF
				0:
					FOR j := 0 TO 23 DO
						tf[j].qds.b.IV := 1;
					END_FOR
		END_CASE
	END_CASE
END_FOR

METHOD Init: BOOL;
VAR_INPUT
END_VAR
VAR

END_VAR
SUPER^.Init();
transaction.typ := RLTM.RLTM_TRANSACTION_TYP_DATA;
transaction.mfc := 3;
transaction.offset := 0;
transaction.len := 46;
transaction.swap_byte := 1;
transaction.pData := ADR(data_real[0]);
transaction.pRes := ADR(res[0]);
transaction.timer.PT := T#1S;
SUPER^.AppendTransaction();

Init := 1;
END_METHOD

END_FUNCTION_BLOCK

// A1_01A/Application/Devices/Pubo_aviogas
FUNCTION_BLOCK Pubo_aviogas EXTENDS RLTM.DeviceTemplate
VAR_INPUT
END_VAR
VAR_OUTPUT
	tf: ARRAY[0..21] OF RLTNU.IEC_M_ME_NC;
END_VAR
VAR
	data_real: ARRAY[0..21] OF REAL;
	res: ARRAY[0..9] OF RLTM.RLTM_MODBUS_TRANSACTION_RESULT;
	i, j: UINT;
	c: ARRAY[0..15] OF UINT := [ 16#1, 16#2, 16#4, 16#8, 16#10, 16#20, 16#40, 16#80, 16#100, 16#200, 16#400, 16#800, 16#1000, 16#2000, 16#4000, 16#8000 ];
END_VAR

(*
Мгновенная активная мощность по фазе 1
Мгновенная активная мощность по фазе 2
Мгновенная активная мощность по фазе 3
Напряжение по фазе 1
Напряжение по фазе 2
Напряжение по фазе 3
Ток по фазе 1
Ток по фазе 2
Ток по фазе 3
Суммарная активная мощность от сброса
Суммарная активная мощность до сброса
Суммарная реактивная мощность от сброса
Суммарная реактивная мощность до сброса
Активная мощность от сброса за текущие сутки
Активная мощность до сброса за текущие сутки
Реактивная мощность от сброса за текущие сутки
Реактивная мощность до сброса за текущие сутки
Активная мощность от сброса за предыдущие сутки
Активная мощность до сброса за предыдущие сутки
Реактивная мощность от сброса за предыдущие сутки
Реактивная мощность до сброса за предыдущие сутки
*)
FOR i := 0 TO 0 DO
	CASE res[i] OF
		RLTM.RLTM_TRANSACTION_RESULT_PROCESSING:
			;//nothing to do
		RLTM.RLTM_TRANSACTION_RESULT_SUCCESS:
			CASE i OF
				0:
					FOR j := 0 TO 21 DO
						tf[j].value := data_real[j];
						tf[j].qds.b.IV := 0;
					END_FOR
				
			END_CASE
	ELSE
		CASE i OF
				0:
					FOR j := 0 TO 21 DO
						tf[j].qds.b.IV := 1;
					END_FOR
		END_CASE
	END_CASE
END_FOR

METHOD Init: BOOL;
VAR_INPUT
END_VAR
VAR

END_VAR
SUPER^.Init();
transaction.typ := RLTM.RLTM_TRANSACTION_TYP_DATA;
transaction.mfc := 3;
transaction.offset := 0;
transaction.len := 42;
transaction.swap_byte := 1;
transaction.pData := ADR(data_real[0]);
transaction.pRes := ADR(res[0]);
transaction.timer.PT := T#1S;
SUPER^.AppendTransaction();

Init := 1;
END_METHOD

END_FUNCTION_BLOCK

// A1_01A/Application/Devices/Istok
FUNCTION_BLOCK Istok EXTENDS RLTM.DeviceTemplate
VAR_INPUT
END_VAR
VAR_OUTPUT
	tf: ARRAY[0..21] OF RLTNU.IEC_M_ME_NC;
END_VAR
VAR
	data_real: ARRAY[0..21] OF REAL;
	res: ARRAY[0..9] OF RLTM.RLTM_MODBUS_TRANSACTION_RESULT;
	i, j: UINT;
	c: ARRAY[0..15] OF UINT := [ 16#1, 16#2, 16#4, 16#8, 16#10, 16#20, 16#40, 16#80, 16#100, 16#200, 16#400, 16#800, 16#1000, 16#2000, 16#4000, 16#8000 ];
END_VAR

(*
Мгновенная активная мощность по фазе 1
Мгновенная активная мощность по фазе 2
Мгновенная активная мощность по фазе 3
Напряжение по фазе 1
Напряжение по фазе 2
Напряжение по фазе 3
Ток по фазе 1
Ток по фазе 2
Ток по фазе 3
Суммарная активная мощность от сброса
Суммарная активная мощность до сброса
Суммарная реактивная мощность от сброса
Суммарная реактивная мощность до сброса
Активная мощность от сброса за текущие сутки
Активная мощность до сброса за текущие сутки
Реактивная мощность от сброса за текущие сутки
Реактивная мощность до сброса за текущие сутки
Активная мощность от сброса за предыдущие сутки
Активная мощность до сброса за предыдущие сутки
Реактивная мощность от сброса за предыдущие сутки
Реактивная мощность до сброса за предыдущие сутки
*)
FOR i := 0 TO 0 DO
	CASE res[i] OF
		RLTM.RLTM_TRANSACTION_RESULT_PROCESSING:
			;//nothing to do
		RLTM.RLTM_TRANSACTION_RESULT_SUCCESS:
			CASE i OF
				0:
					FOR j := 0 TO 21 DO
						tf[j].value := data_real[j];
						tf[j].qds.b.IV := 0;
					END_FOR
				
			END_CASE
	ELSE
		CASE i OF
				0:
					FOR j := 0 TO 21 DO
						tf[j].qds.b.IV := 1;
					END_FOR
		END_CASE
	END_CASE
END_FOR

METHOD Init: BOOL;
VAR_INPUT
END_VAR
VAR

END_VAR
SUPER^.Init();
transaction.typ := RLTM.RLTM_TRANSACTION_TYP_DATA;
transaction.mfc := 3;
transaction.offset := 0;
transaction.len := 42;
transaction.swap_byte := 1;
transaction.pData := ADR(data_real[0]);
transaction.pRes := ADR(res[0]);
transaction.timer.PT := T#1S;
SUPER^.AppendTransaction();

Init := 1;
END_METHOD

END_FUNCTION_BLOCK

// A1_01A/Application/Devices/Datacom
FUNCTION_BLOCK Datacom EXTENDS RLTM.DeviceTemplate
VAR_INPUT
END_VAR
VAR_OUTPUT
	tf: ARRAY[0..21] OF RLTNU.IEC_M_ME_NC;
END_VAR
VAR
	data_real: ARRAY[0..21] OF REAL;
	res: ARRAY[0..9] OF RLTM.RLTM_MODBUS_TRANSACTION_RESULT;
	i, j: UINT;
	c: ARRAY[0..15] OF UINT := [ 16#1, 16#2, 16#4, 16#8, 16#10, 16#20, 16#40, 16#80, 16#100, 16#200, 16#400, 16#800, 16#1000, 16#2000, 16#4000, 16#8000 ];
END_VAR

(*
Давление
Температура
Абсолютное давление
Коэффициент коррекции 
Коэффициент сжимаемости газа
Содержание азота
Содержание водорода
Содержание двуокиси углерода
Плость газа при нормальных условиях
Рабочий расход газа
Стандартный расход газа
Мощность
Теплотворная способность
Коэффициент плотности
Давление
Температура
Рабочий объём
Стандартный объём
Энергия
Рабочий расход прошлые сутки
Стандартный расход прошлые сутки
Рабочий расход прошлый месяц
Стандартный расход прошлый месяц
*)
FOR i := 0 TO 0 DO
	CASE res[i] OF
		RLTM.RLTM_TRANSACTION_RESULT_PROCESSING:
			;//nothing to do
		RLTM.RLTM_TRANSACTION_RESULT_SUCCESS:
			CASE i OF
				0:
					FOR j := 0 TO 23 DO
						tf[j].value := data_real[j];
						tf[j].qds.b.IV := 0;
					END_FOR
				
			END_CASE
	ELSE
		CASE i OF
				0:
					FOR j := 0 TO 23 DO
						tf[j].qds.b.IV := 1;
					END_FOR
		END_CASE
	END_CASE
END_FOR

METHOD Init: BOOL;
VAR_INPUT
END_VAR
VAR

END_VAR
SUPER^.Init();
transaction.typ := RLTM.RLTM_TRANSACTION_TYP_DATA;
transaction.mfc := 3;
transaction.offset := 0;
transaction.len := 46;
transaction.swap_byte := 1;
transaction.pData := ADR(data_real[0]);
transaction.pRes := ADR(res[0]);
transaction.timer.PT := T#1S;
SUPER^.AppendTransaction();

Init := 1;
END_METHOD

END_FUNCTION_BLOCK

// Server_TCP/Server_group
FUNCTION_BLOCK Server_group
VAR_INPUT
END_VAR
VAR
	servers			: POINTER TO Server;	
	servers_qnt		: UINT;
	i				: UINT;
END_VAR

IF (servers = 0) THEN
	RETURN;
END_IF

FOR i := 0 TO servers_qnt - 1 DO
	ServerRun(ADR(servers[i]));
END_FOR

METHOD Init : BOOL
VAR_INPUT
	serversCfg		: POINTER TO ServerCfg;
	clientsCfg		: POINTER TO ClientCfg;
	ip2rs_buffer	: POINTER TO Exchange_Buffer;
END_VAR
VAR
	i			: UINT;
	result		: RTS_IEC_RESULT;
	address		: SOCKADDRESS;
	init_res	: BOOL;
	name		: STRING;
END_VAR
servers := 0;

IF (serversCfg = 0) OR (clientsCfg = 0) OR (ip2rs_buffer = 0) THEN
	Init := FALSE;
	RETURN;
END_IF


i := 0;
WHILE (LEN(serversCfg[i].address)>0) AND (i < SERVER_MAX_COUNT) DO
	i := i+1;
END_WHILE

IF i = 0 THEN
	Init := FALSE;
	RETURN;
END_IF

servers_qnt := i;
name := UDINT_TO_STRING(THIS);
servers := SysMemAllocData(name, servers_qnt*SIZEOF(Server), ADR(result));
IF servers = 0 THEN
	Init := FALSE;
	RETURN;
END_IF

SysMemSet(servers, 0, servers_qnt*SIZEOF(Server));
FOR i := 0 TO servers_qnt - 1 DO
		
	address.sin_family := SOCKET_AF_INET;
	address.sin_port := SysSockHtons(serversCfg[i].port);
	result := SysSockInetAddr(serversCfg[i].address, ADR(address.sin_addr.ulAddr));
	IF result <> CmpErrors.Errors.ERR_OK THEN
		Init := FALSE;
		fb_exit(FALSE);
		RETURN;
	END_IF
	
	init_res := ServerInit(srv := ADR(servers[i]), address := address, socket_type := serversCfg[i].socket_type, max_connections := serversCfg[i].max_connections, clients_cfg := clientsCfg, ip2rs := ip2rs_buffer);
	IF init_res = FALSE THEN
		Init := FALSE;
		fb_exit(FALSE);
		RETURN;
	END_IF

END_FOR

Init := TRUE;
END_METHOD

METHOD ServerRun
VAR_INPUT
	srv : POINTER TO Server;
END_VAR
VAR
	client_address		: SOCKADDRESS;
	size				: UDINT;
	result				: RTS_IEC_RESULT;
	client_socket		: SysSocket.RTS_IEC_HANDLE;
	i, count			: UINT;
	client_index		: INT;
	client_cfg			: POINTER TO ClientCfg;	
	fdRead				: SOCKET_FD_SET;
	fdExcept			: SOCKET_FD_SET;
	timeout				: SOCKET_TIMEVAL;
	diReady				: DINT;	
	numberofbytes		:__XINT;
	tx_length			: UINT;
	need_tx				: BOOL;
	state				: UINT;
END_VAR
IF (srv = 0) THEN
	RETURN;
END_IF

IF srv^.socket = 0 THEN
	srv^.socket := SysSockCreate(SOCKET_AF_INET, SOCKET_STREAM, SOCKET_IPPROTO_TCP, ADR(result));
	IF (srv^.socket = SysSocket.RTS_INVALID_HANDLE) THEN RETURN; END_IF
	result := SysSockBind(srv^.socket, ADR(srv^.address), SIZEOF(SOCKADDRESS));	// 1 - Bind
	IF (result = CmpErrors.Errors.ERR_OK) THEN
		result := SysSockListen(srv^.socket, srv^.max_connections);													// 2 - Listen
	END_IF
	IF (result <> CmpErrors.Errors.ERR_OK) THEN
		SysSockClose(srv^.socket);
		srv^.socket := 0;
		RETURN;
	END_IF
END_IF

size := SIZEOF(client_address);
client_socket := SysSockAccept(srv^.socket, ADR(client_address), ADR(size), ADR(result));
IF (result = CmpErrors.Errors.ERR_OK) THEN
	
	client_index := GetFreeClientIndex(srv);
	client_cfg := GetClientConfig(srv^.clients_cfg, client_address.sin_addr.ulAddr, srv^.address.sin_port);
		
	IF (client_index < 0) OR (client_cfg = 0) THEN
		SysSockClose(client_socket);
	ELSE
		srv^.clients[client_index].socket := client_socket;
		srv^.clients[client_index].address := client_address;
		srv^.clients[client_index].rs_port := client_cfg^.rs_port;
		srv^.clients[client_index].ttl := 0;
		srv^.ip2rs_buffer^.AddIPMessage(srv^.address.sin_port, srv^.clients[client_index].address.sin_addr.ulAddr, srv^.clients[client_index].rs_port, OPEN_CONNECTION, ADR(srv^.rx_data), 0);		
	END_IF
END_IF


FOR i := 0 TO srv^.max_connections - 1 DO
	IF srv^.clients[i].socket <> 0 THEN		
	//	srv^.clients[i].ttl();
	//	IF srv^.clients[i].ttl.Q THEN			
	//	ClientClose(srv, i);	
	//	END_IF
	END_IF
END_FOR

SysSockFdZero(fdRead);
SysSockFdZero(fdExcept);

FOR i := 0 TO srv^.max_connections - 1 DO
	IF srv^.clients[i].socket <> 0 THEN		
		count := srv^.ip2rs_buffer^.CheckIPMessage(srv^.address.sin_port, srv^.clients[i].address.sin_addr.ulAddr, srv^.clients[i].rs_port);		
		IF (count = 0) THEN
			SysSockFdInit(srv^.clients[i].socket, fdRead);
		END_IF
		SysSockFdInit(srv^.clients[i].socket, fdExcept);
	END_IF
END_FOR

timeout.tv_sec := 0;
timeout.tv_usec := 0;
	
result := SysSockSelect( srv^.max_connections, ADR(fdRead), 0, ADR(fdExcept), ADR(timeout), ADR(diReady)); 
IF (result = CmpErrors.Errors.ERR_OK) AND (diReady <> 0) THEN

	FOR i := 0 TO srv^.max_connections - 1 DO
		IF srv^.clients[i].socket = 0 THEN	CONTINUE; END_IF

		IF SysSockFdIsset(srv^.clients[i].socket, fdExcept) THEN
			ClientClose(srv, i);
		ELSIF SysSockFdIsset(srv^.clients[i].socket, fdRead) THEN
			
			numberOfBytes := SysSockRecv(srv^.clients[i].socket, ADR(srv^.rx_data), SIZEOF(srv^.rx_data), 0, ADR(result));

			IF (result <> CmpErrors.Errors.ERR_OK AND result <> CmpErrors.Errors.ERR_SOCK_WOULDBLOCK) THEN				
				ClientClose(srv, i);			
			ELSIF (numberOfBytes <> 0) THEN
				srv^.ip2rs_buffer^.AddIPMessage(srv^.address.sin_port, srv^.clients[i].address.sin_addr.ulAddr, srv^.clients[i].rs_port, WORK_CONNECTION, ADR(srv^.rx_data), DINT_TO_UINT(numberOfBytes));
			END_IF
		END_IF
	END_FOR
END_IF

FOR i := 0 TO srv^.max_connections - 1 DO
	IF srv^.clients[i].socket <> 0 THEN			
		need_tx := srv^.ip2rs_buffer^.GetMessageForIP(srv^.address.sin_port, srv^.clients[i].address.sin_addr.ulAddr, srv^.clients[i].rs_port, ADR(state), ADR(srv^.tx_data), SIZEOF(srv^.tx_data), ADR(tx_length));
		IF (need_tx) THEN
			CASE (state) OF		
				WORK_CONNECTION:
					numberofbytes := SysSockSend(srv^.clients[i].socket, ADR(srv^.tx_data), tx_length, 0, ADR(result));
					IF (result <> CmpErrors.Errors.ERR_OK AND result <> CmpErrors.Errors.ERR_SOCK_WOULDBLOCK) THEN
						ClientClose(srv, i);			
					END_IF
				CLOSE_CONNECTION:
				//	ClientClose(srv, i);			
					SysSockClose(srv^.clients[i].socket);
					srv^.clients[i].socket := 0;
					srv^.ip2rs_buffer^.ClearByClient(srv^.address.sin_port, srv^.clients[i].address.sin_addr.ulAddr, srv^.clients[i].rs_port);
					srv^.clients[i].ttl := 0;
			END_CASE			
		END_IF
	END_IF
END_FOR
END_METHOD

METHOD ServerInit : BOOL
VAR_INPUT
	srv				: POINTER TO Server;	// 	
	address			: SOCKADDRESS;			//
	socket_type		: DINT;					// SOCKET_STREAM, SOCKET_DGRAM
	max_connections : UINT;					//
	clients_cfg		: POINTER TO ClientCfg;	// 
	ip2rs			: POINTER TO Exchange_Buffer;	//
END_VAR
VAR
	i		: UINT;
	result : RTS_IEC_RESULT;
	name	: STRING;
END_VAR

IF (srv = 0) OR (clients_cfg = 0) OR (ip2rs = 0) OR (max_connections = 0) OR (max_connections > SERVER_MAX_CONNECTIONS) OR (socket_type <> SOCKET_STREAM AND socket_type <> SOCKET_DGRAM) THEN
	ServerInit := FALSE;
	RETURN;
END_IF

srv^.max_connections := max_connections;
srv^.socket_type := socket_type;
srv^.address := address;
srv^.clients_cfg := clients_cfg;
srv^.ip2rs_buffer := ip2rs;

name := UDINT_TO_STRING(srv);
srv^.clients := SysMemAllocData(name, max_connections*SIZEOF(SClient), ADR(result));
IF srv^.clients = 0 THEN
	ServerInit := FALSE;
	RETURN;
END_IF

SysMemSet(srv^.clients, 0, max_connections*SIZEOF(SClient));
srv^.socket := 0;

ServerInit := TRUE;
END_METHOD

METHOD ServerDeinit
VAR_INPUT
	srv				: POINTER TO Server;	// 	
END_VAR
VAR
	i		: UINT;
	result	: RTS_IEC_RESULT;
	name	: STRING;
END_VAR

IF (srv = 0) THEN
	RETURN;
END_IF

IF srv^.clients <> 0 THEN	
	FOR i := 0 TO srv^.max_connections - 1 DO		
		IF srv^.clients[i].socket <> 0 THEN 
			SysSockClose(srv^.clients[i].socket);
			srv^.clients[i].socket := 0;
		END_IF;		
	END_FOR
	name := UDINT_TO_STRING(srv);
	SysMemFreeData(name, srv^.clients);
	srv^.clients := 0;	
END_IF

IF srv^.socket <> 0 THEN 
	SysSockClose(srv^.socket);
	srv^.socket := 0;
END_IF;
END_METHOD

METHOD fb_exit : BOOL
VAR_INPUT
	bInCopyCode : BOOL; // if TRUE, the exit method is called for exiting an instance that is copied afterwards (online change). 
END_VAR
VAR
	i		: UINT;
	result	: RTS_IEC_RESULT;
	name	: STRING;
END_VAR

IF (servers = 0) THEN
	RETURN;
END_IF

FOR i := 0 TO servers_qnt - 1 DO
	ServerDeinit(ADR(servers[i]));
END_FOR

name := UDINT_TO_STRING(THIS);
SysMemFreeData(name, servers);
servers := 0;
END_METHOD

METHOD fb_init : BOOL
VAR_INPUT
	bInitRetains : BOOL; // if TRUE, the retain variables are initialized (warm start / cold start)
	bInCopyCode : BOOL;  // if TRUE, the instance afterwards gets moved into the copy code (online change)

//	serversCfg		: POINTER TO ServerCfg;
//	clientsCfg		: POINTER TO ClientCfg;
	//ip2rs_buffer	: POINTER TO Exchange_Buffer;
END_VAR
VAR
	i			: UINT;
	result		: RTS_IEC_RESULT;
	address		: SOCKADDRESS;
	init_res	: BOOL;
	name		: STRING;
END_VAR
(*servers := 0;

IF (serversCfg = 0) OR (clientsCfg = 0) OR (ip2rs_buffer = 0) THEN
	fb_init := FALSE;
	RETURN;
END_IF


i := 0;
WHILE (LEN(serversCfg[i].address)>0) AND (i < SERVER_MAX_QOUNT) DO
	i := i+1;
END_WHILE

IF i = 0 THEN
	fb_init := FALSE;
	RETURN;
END_IF

servers_qnt := i;
name := UDINT_TO_STRING(THIS);
servers := SysMemAllocData(name, servers_qnt*SIZEOF(Server), ADR(result));
IF servers = 0 THEN
	fb_init := FALSE;
	RETURN;
END_IF

SysMemSet(servers, 0, servers_qnt*SIZEOF(Server));
FOR i := 0 TO servers_qnt - 1 DO
		
	address.sin_family := SOCKET_AF_INET;
	address.sin_port := SysSockHtons(serversCfg[i].port);
	result := SysSockInetAddr(serversCfg[i].address, ADR(address.sin_addr.ulAddr));
	IF result <> CmpErrors.Errors.ERR_OK THEN
		fb_init := FALSE;
		fb_exit(FALSE);
		RETURN;
	END_IF
	
	init_res := ServerInit(srv := ADR(servers[i]), address := address, socket_type := serversCfg[i].socket_type, max_connections := serversCfg[i].max_connections, clients_cfg := clientsCfg, ip2rs := ip2rs_buffer);
	IF init_res = FALSE THEN
		fb_init := FALSE;
		fb_exit(FALSE);
		RETURN;
	END_IF

END_FOR

fb_init := TRUE;
*)
END_METHOD

METHOD GetFreeClientIndex : INT
VAR_INPUT
	srv : POINTER TO Server;
END_VAR
VAR
	i	: UINT;
END_VAR
GetFreeClientIndex := -1;

IF (srv = 0) THEN
	RETURN;
END_IF

FOR i := 0 TO srv^.max_connections - 1 DO
	IF srv^.clients[i].socket = 0 THEN
		GetFreeClientIndex := i; 
		RETURN;
	END_IF
END_FOR
END_METHOD

METHOD GetClientConfig : POINTER TO ClientCfg
VAR_INPUT
	clients_cfg		: POINTER TO ClientCfg;	//
	client_address	: UDINT;
	server_port		: UINT; 
END_VAR
VAR
	i, port : UINT;
	address	: UDINT;	
	result : RTS_IEC_RESULT;
END_VAR
GetClientConfig := 0;
i := 0;

IF (clients_cfg = 0) THEN
	RETURN;
END_IF

WHILE LEN(clients_cfg[i].client_address) > 0 DO
	result := SysSockInetAddr(clients_cfg[i].client_address, ADR(address));
	IF result <> CmpErrors.Errors.ERR_OK THEN
		RETURN;
	END_IF	
	port := SysSockHtons(clients_cfg[i].server_port);	
	IF (address = client_address) AND (port = server_port) THEN
		GetClientConfig := ADR(clients_cfg[i]);
		RETURN;
	END_IF	
	i := i+1;
END_WHILE
END_METHOD

METHOD ClientClose
VAR_INPUT
	srv			: POINTER TO Server;
	client_i	: UINT;
END_VAR
VAR
END_VAR
IF (srv = 0) OR (client_i >= srv^.max_connections) THEN
	RETURN;
END_IF

IF srv^.clients[client_i].socket <> 0 THEN		
	SysSockClose(srv^.clients[client_i].socket);
	srv^.clients[client_i].socket := 0;
	srv^.ip2rs_buffer^.ClearByClient(srv^.address.sin_port, srv^.clients[client_i].address.sin_addr.ulAddr, srv^.clients[client_i].rs_port);
	srv^.ip2rs_buffer^.AddIPMessage(srv^.address.sin_port, srv^.clients[client_i].address.sin_addr.ulAddr, srv^.clients[client_i].rs_port, CLOSE_CONNECTION, ADR(srv^.rx_data), 0);
	SysMemSet(ADR(srv^.clients[client_i].address), 0, SIZEOF(srv^.clients[client_i].address));
	srv^.clients[client_i].rs_port := 0;
	srv^.clients[client_i].ttl := 0;
END_IF
END_METHOD

END_FUNCTION_BLOCK
